(**************************************************************************************
 * 	Application		:	BoxControl Framework
 *	Revision		:	$Revision: 404529 $
 *	Revision date	:	$Date: 2018-04-23 08:21:38 +0200 (Mo., 23 Apr 2018) $
 *	Last changed by	:	$Author: b7bolm $
 *	URL				:	$URL: http://almscdc.swisslog.com/repo/SWPD/Development/BoxControlFramework/20_Release/trunk/01_Software/BCF/BCF/JumpStart/20_Product/10_App/10_Base/10_Lib/00_GVLs/GVR_Table.TcGVL $
 *
 *	Purpose			:	GVR signals - Separated due to debug reasons.
 *
 * ------------------------------------------------------------------------------------
 *	Copyright Swisslog [IP AG], Switzerland. All rights reserved.
 * 
 * ------------------------------------------------------------------------------------
 *	
 * 	Revision History: 
 *
 * 	VERSION			DATE			INITIALS			DESCRIPTION
 *	0.1				01.01.2001		swl					Example
 *
 **************************************************************************************)

VAR_GLOBAL CONSTANT
	NUMBER_OF_GVR_SIGNALS			: INT := 9999; // Number of ISR signals, max 9999 
END_VAR
 
VAR_GLOBAL
	GlobalVariable					: ARRAY[0..NUMBER_OF_GVR_SIGNALS, 0..9] OF DINT; // Array for GVR telegram
END_VAR

(* stored: Version 1.1.0.1, ProductVersion 3.1.4022.12
   GVL GVR_Table: Id {f012601b-ed54-48ce-bcb6-0afc6c8573b0} *)
